PROGRAM prgComEffIO
VAR
	fbCom		: FB_MqttCommunicator_V2;
END_VAR

fbCom(
	bConnect				:= TRUE,
	strAuthKey				:= 'EIO08031879806', 
	sUserName				:= '825f07c4-bbac-469f-beae-0c4ad006bf93', 
	sUserPassword			:= 'b1111145-4452-4020-8dff-f640d68312f3', 
	eSavePositionCertificate:= eSavePositionOnPLC.ePostionC, 
	bConnected=> , 
	bError=> , 
	hrErrorCode=> , 
	eConnectionState=> , 
	eErrorMessage_Out=> );

END_PROGRAM

(* stored: Version 1.1.0.1, ProductVersion 3.1.4024.11
   POU prgComEffIO: Id {cbcd318b-bf51-484c-bcaa-d6efcdf43fe3}, SpecialFunc None *)
